Fanuc KAREL source: port_RDO.kl

PROGRAM TP
%NOLOCKGROUP
VAR
 x: BOOLEAN
BEGIN
 x = RDO[3]
END TP
